// Mitsubishi GX Works2 project: OR   PLC: Q03UDV

PROGRAM MAIN
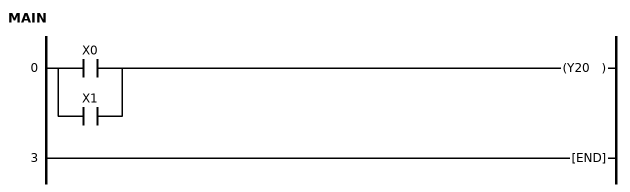
0     LD      X0
      OR      X1
      OUT     Y20
3     END
END_PROGRAM
